Universal Robots URScript: step4e_detached_movel_minrot_v21.script

# Step4e P1-a detached movel minimal-rotation v21.
# VERSION: 2026-06-11T1601HKT_STEP4E_DETACHED_MOVEL_MINROT_V21
# GENERATED_AT_LOCAL: 2026-06-11T16:01:43+08:00
# PURPOSE: latch first contact normal, detach along the locked normal, then preview the minimal-rotation target without contact-posture motion.
# CONTROL: bridge step4e-version=v21 writes 37..39 as +locked-normal detach direction in 25.1 and 40..42 as target rotvec for z_tcp_B ~= -locked_normal_B in 25.2.
# SAFETY: raw normal guard 35 N, force norm guard 50 N, torque guard 3.0 Nm.

def codex_abs(x):
  if x < 0.0:
    return -x
  end
  return x
end

def codex_clamp(x, lo, hi):
  if x < lo:
    return lo
  elif x > hi:
    return hi
  end
  return x
end

def codex_wait_for_fresh_heartbeat(timeout_s):
  local t = 0.0
  local initial_heartbeat = read_input_float_register(26)
  local current_heartbeat = initial_heartbeat
  while t < timeout_s:
    current_heartbeat = read_input_float_register(26)
    write_output_float_register(26, current_heartbeat)
    if read_input_float_register(27) > 0.5 and current_heartbeat != initial_heartbeat:
      return True
    end
    sync()
    t = t + get_steptime()
  end
  return False
end

def codex_wait_for_rezero_complete(timeout_s):
  local t = 0.0
  local initial_heartbeat = read_input_float_register(26)
  local current_heartbeat = initial_heartbeat
  local saw_sensor_not_ready = False
  while t < timeout_s:
    current_heartbeat = read_input_float_register(26)
    write_output_float_register(26, current_heartbeat)
    if read_input_float_register(27) < 0.5:
      saw_sensor_not_ready = True
    elif saw_sensor_not_ready and read_input_float_register(27) > 0.5 and current_heartbeat != initial_heartbeat:
      return True
    end
    sync()
    t = t + get_steptime()
  end
  return False
end

def codex_step4e_guard_stop_reason():
  local normal_force = read_input_float_register(24)
  local force_norm = read_input_float_register(25)
  local sensor_ok = read_input_float_register(27)
  local stop_request = read_input_float_register(28)
  local torque_norm = read_input_float_register(30)
  if sensor_ok < 0.5:
    return 3.0
  elif stop_request > 0.5:
    return 4.0
  elif codex_abs(normal_force) > 35.0:
    return 5.0
  elif force_norm > 50.0:
    return 6.0
  elif torque_norm > 3.0:
    return 7.0
  end
  return 0.0
end

def codex_should_auto_home(stop_reason):
  if stop_reason == 1.0:
    return True
  elif stop_reason == 2.0:
    return True
  elif stop_reason == 4.0:
    return True
  elif stop_reason == 5.0:
    return True
  elif stop_reason == 6.0:
    return True
  elif stop_reason == 7.0:
    return True
  elif stop_reason == 8.0:
    return True
  elif stop_reason == 9.0:
    return True
  elif stop_reason == 10.0:
    return True
  elif stop_reason == 12.0:
    return True
  elif stop_reason == 13.0:
    return True
  elif stop_reason == 14.0:
    return True
  end
  return False
end

def codex_echo_basic(stop_reason):
  write_output_float_register(24, read_input_float_register(24))
  write_output_float_register(25, read_input_float_register(25))
  write_output_float_register(26, read_input_float_register(26))
  write_output_float_register(27, read_input_float_register(27))
  write_output_float_register(28, read_input_float_register(28))
  write_output_float_register(29, read_input_float_register(29))
  write_output_float_register(30, stop_reason)
end

def codex_echo_step4e(stop_reason):
  codex_echo_basic(stop_reason)
  write_output_float_register(31, read_input_float_register(44))
  write_output_float_register(32, read_input_float_register(45))
  write_output_float_register(33, read_input_float_register(39))
  write_output_float_register(36, read_input_float_register(37))
  write_output_float_register(37, read_input_float_register(38))
  write_output_float_register(38, read_input_float_register(39))
  write_output_float_register(39, read_input_float_register(40))
  write_output_float_register(40, read_input_float_register(41))
  write_output_float_register(41, read_input_float_register(42))
  write_output_float_register(42, read_input_float_register(43))
  write_output_float_register(43, read_input_float_register(44))
  write_output_float_register(44, read_input_float_register(45))
  write_output_float_register(45, read_input_float_register(46))
  write_output_float_register(46, read_input_float_register(47))
end


def codex_wait_for_cmd_valid(stage_code, timeout_s):
  local t = 0.0
  local last_heartbeat = read_input_float_register(26)
  local stale_s = 0.0
  while t < timeout_s:
    write_output_float_register(35, stage_code)
    local heartbeat = read_input_float_register(26)
    if heartbeat == last_heartbeat:
      stale_s = stale_s + get_steptime()
    else:
      stale_s = 0.0
      last_heartbeat = heartbeat
    end
    codex_echo_step4e(0.0)
    if stale_s > 0.100:
      return 2.0
    end
    local guard_reason = codex_step4e_guard_stop_reason()
    if guard_reason != 0.0:
      return guard_reason
    end
    if read_input_float_register(43) >= 0.5:
      return 0.0
    end
    sync()
    t = t + get_steptime()
  end
  return 12.0
end

def codex_step4e_detached_movel_v21():
  local stop_reason = 0.0
  local home_pose = get_actual_tcp_pose()
  local search_accel_m_s2 = 0.300
  local search_hold_s = 0.002
  local stale_limit_s = 0.100
  local search_runtime_limit_s = 40.0
  local search_near_start_depth_m = 0.080
  local max_search_down_m = 0.092
  local search_far_speed_m_s = -0.015
  local search_near_speed_m_s = -0.003
  local contact_triggered = 0
  textmsg("codex step4e version 2026-06-11T1601HKT_STEP4E_DETACHED_MOVEL_MINROT_V21 start detached_movel_v21")
  write_output_float_register(34, 0.0)
  write_output_float_register(35, 20.0)
  codex_echo_step4e(0.0)
  if not codex_wait_for_fresh_heartbeat(30.0):
    stop_reason = 3.0
  end
  if stop_reason == 0.0:
    write_output_float_register(35, 22.0)
    local p1 = get_actual_tcp_pose()
    local entry_pose = p[0.433010000, 0.108020000, p1[2], 3.141592654, 0.0, 0.0]
    movel(entry_pose, a=0.030, v=0.020, r=0.0)
    stopl(0.1)
    write_output_float_register(35, 23.0)
    codex_echo_step4e(stop_reason)
    write_output_float_register(34, 1.0)
    if not codex_wait_for_rezero_complete(5.0):
      stop_reason = 14.0
    end
  end
  if stop_reason == 0.0:
    write_output_float_register(35, 24.0)
    local search_start = get_actual_tcp_pose()
    local last_heartbeat = read_input_float_register(26)
    local stale_s = 0.0
    local t = 0.0
    while stop_reason == 0.0:
      local heartbeat = read_input_float_register(26)
      local normal_force = read_input_float_register(24)
      local force_norm = read_input_float_register(25)
      local pose_now = get_actual_tcp_pose()
      local search_depth_m = search_start[2] - pose_now[2]
      if heartbeat == last_heartbeat:
        stale_s = stale_s + get_steptime()
      else:
        stale_s = 0.0
        last_heartbeat = heartbeat
      end
      if normal_force <= -1.0 or force_norm > 1.5:
        contact_triggered = 1
        stop_reason = 11.0
      elif stale_s > stale_limit_s:
        stop_reason = 2.0
      else:
        stop_reason = codex_step4e_guard_stop_reason()
      end
      if stop_reason == 0.0:
        if search_depth_m >= max_search_down_m:
          stop_reason = 8.0
        elif t >= search_runtime_limit_s:
          stop_reason = 10.0
        else:
          if search_depth_m < search_near_start_depth_m:
            codex_echo_step4e(stop_reason)
            speedl([0.0, 0.0, search_far_speed_m_s, 0.0, 0.0, 0.0], search_accel_m_s2, search_hold_s)
          else:
            write_output_float_register(35, 24.2)
            codex_echo_step4e(stop_reason)
            speedl([0.0, 0.0, search_near_speed_m_s, 0.0, 0.0, 0.0], search_accel_m_s2, search_hold_s)
          end
          t = t + get_steptime()
        end
      end
    end
    stopl(0.1)
  end
  if contact_triggered == 1:
    stop_reason = 0.0
  end
  if stop_reason == 0.0:
    write_output_float_register(35, 25.05)
    stop_reason = codex_wait_for_cmd_valid(25.05, 1.000)
  end
  if stop_reason == 0.0:
    write_output_float_register(35, 25.1)
    stop_reason = codex_wait_for_cmd_valid(25.1, 1.000)
    local detach_total_m = 0.0
    while stop_reason == 0.0 and detach_total_m < 0.002 and read_input_float_register(25) > 2.0:
      local dir_x = read_input_float_register(37)
      local dir_y = read_input_float_register(38)
      local dir_z = read_input_float_register(39)
      local step_m = 0.001
      local p_detach = get_actual_tcp_pose()
      local detach_pose = p[p_detach[0] + step_m * dir_x, p_detach[1] + step_m * dir_y, p_detach[2] + step_m * dir_z, p_detach[3], p_detach[4], p_detach[5]]
      codex_echo_step4e(stop_reason)
      movel(detach_pose, a=0.030, v=0.010, r=0.0)
      stopl(0.1)
      detach_total_m = detach_total_m + step_m
      stop_reason = codex_step4e_guard_stop_reason()
    end
  end
  if stop_reason == 0.0:
    write_output_float_register(35, 25.2)
    stop_reason = codex_wait_for_cmd_valid(25.2, 1.000)
    if stop_reason == 0.0:
      # 25.2 is target-preview only; no contact-posture movel.
      codex_echo_step4e(stop_reason)
      sleep(0.250)
      if read_input_float_register(46) > 0.030:
        stop_reason = 15.0
      else:
        stop_reason = codex_step4e_guard_stop_reason()
      end
    end
  end
  if stop_reason == 15.0 or codex_should_auto_home(stop_reason):
    write_output_float_register(35, 27.0)
    codex_echo_step4e(stop_reason)
    movel(home_pose, a=0.030, v=0.020, r=0.0)
    stopl(0.1)
  end
  write_output_float_register(30, stop_reason)
  write_output_float_register(35, 29.0)
  textmsg("codex step4e version 2026-06-11T1601HKT_STEP4E_DETACHED_MOVEL_MINROT_V21 stop reason:", stop_reason)
end

codex_step4e_detached_movel_v21()
